# EPICS SNL sequencer program: acq400iocApp/src/autoRepeat.stt
/*************************************************************************\
autoRepeat.st : repeat transient on termination
\*************************************************************************/
program autoRepeat
option +r;

int tstate;
assign tstate to "{uut}:MODE:TRANS_ACT:STATE";
monitor tstate;

int repeat;
assign repeat to "{uut}:MODE:TRANSIENT:REPEAT";
monitor repeat;

int set_arm;
assign set_arm to "{uut}:MODE:TRANSIENT:SET_ARM";

int repeat_delay_ms;
assign repeat_delay_ms to "{uut}:MODE:TRANSIENT:DELAYMS";

double repeat_delay;

int set_abort;
assign set_abort to "{uut}:MODE:TRANSIENT:SET_ABORT";
monitor set_abort;

int shot_complete;
assign shot_complete to "{uut}:SHOT_COMPLETE";
monitor shot_complete;

int shot_complete0;

int continuous;
assign continuous to "{uut}:MODE:CONTINUOUS";
monitor continuous;

%{
#include <sys/types.h>
#include <sys/stat.h>
#include <fcntl.h>
#include <stdlib.h>
#include <unistd.h>

int fd = 1;

void openDebug(char* debug){
	if (debug == 0 || debug[0] == '\0'){
		fd = 1;
	}else{
		fd = open(debug, (O_CREAT | O_WRONLY), 0664);
		if (fd < 0){
			printf("ERROR failed to open debug:%s\n", debug);
			exit(-1);
		}
	}
}

void closeDebug() {
	if (fd != 1) close(fd);
}
}%
ss autorepeat
{
	state init {
		when() {
				openDebug(macValueGet("debug"));
		} state stop
	}

	state stop
	{
		when(tstate != 0){
			printf("stop=>run\n");
		} state run
	}

	state run
	{
		when(set_abort > 0){
			set_abort = 0;
			pvPut(set_abort);
			dprintf(fd, "run=>stop_transition ABORT\n");
		} state stop_transition

		when(tstate == 0){
			dprintf(fd, "run=>run_transition\n");
		} state run_transition
	}

	state stop_transition
	{
		when(tstate == 0){
			dprintf(fd, "stop_transition=>stop\n");
		} state stop
	}

	state run_transition
	{
		when(repeat < 0){
			dprintf(fd, "run_transition=>rearm autorepeat forever\n");
		} state rearm

		when(repeat > 1){
			repeat -= 1;
			pvPut(repeat);
			dprintf(fd, "run_transition=>rearm autorepeat %d\n", repeat);
		} state rearm

		when (repeat == 1){
			repeat = 0;
			pvPut(repeat);
			dprintf(fd, "run_transition=>stop autorepeat finished\n");
		} state stop

		when (repeat == 0){
			dprintf(fd, "run_transition=>stop autorepeat 0\n");
		} state stop
	}

	state rearm
	{
		entry {
      			pvGet(repeat_delay_ms);
      			repeat_delay = repeat_delay_ms/1000;
      			pvGet(shot_complete);
      			shot_complete0 = shot_complete;
    		}
		when(set_abort > 0){
			pvPut(set_abort);
			set_abort = 0;
			dprintf(fd, "run=>stop_transition ABORT\n");
		} state stop_transition

		when (delay(repeat_delay)) {
			dprintf(fd, "rearm=>waitrun\n");
			set_arm = 1;
			pvPut(set_arm);
		} state waitrun
	}

	state waitrun
	{
		when(shot_complete != shot_complete0 && tstate == 0){
			dprintf(fd, "wait_run->run_transition\n");
		} state run_transition

		when(tstate != 0){
			dprintf(fd, "wait_run=>run\n");
		} state run
	}
}

/* avoid spurious restart last transient repeat when continuous is stopped */

ss monitor_continuous
{
	state mc1
	{
		when(continuous > 0){
			pvGet(repeat);
			if (repeat){
				dprintf(fd, "continuous start detected, set repeat to zero to false restart\n");
				repeat = 0;
				pvPut(repeat);
			}
		} state mc2
	}

	state mc2
	{
		when(continuous == 0){
			;
		} state mc1
	}
}

exit
{
	closeDebug();
}
